ABB RobotStudio station: 4230.rsstn

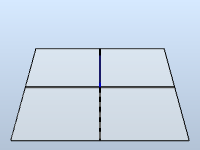
Station Station (saved by RobotStudio 6.7.7936.1011)
Layout (positions relative to the parent item):
